(* CODESYS project lab1.project

Project tree, tasks and I/O mapping:
  Device : CODESYS Control Win V3, 3S - Smart Software Solutions GmbH, order no. 305021, version 3.5.5.50
    application Application
      libraries: Standard, * (System)
      task MainTask (cyclic, interval t#400ms, priority 1) calls task_relay
      task VISU_TASK (cyclic, interval 100 ms, priority 31) calls VisuElems.Visu_Prg
      program task_relay [ST]
      global variables GVL
      visualisation Visualization
  text list GlobalTextList
*)

// Device/Application/GVL
VAR_GLOBAL
	tempeture_sensor: INT := 20;
	door: BOOL := FALSE; // FALSE--> closed ; TRUE --> open
	
//	valve_prop: INT := -24; // FALSE--> closed ; TRUE --> open
//	btn: BOOL := FALSE; // FALSE--> closed ; TRUE --> open
//	btn_peiod: BOOL := FALSE; // FALSE--> closed ; TRUE --> open
END_VAR

// Device/Application/task_relay
PROGRAM task_relay
VAR
	DOOR_LIMIT: INT := 28;
	MIN_VALUE: INT := 15;
	MAX_VALUE: INT := 40;
	MIN_LIMIT: INT;
END_VAR

IF tempeture_sensor > DOOR_LIMIT THEN
	door:= TRUE;
ELSE door:= FALSE;
END_IF

END_PROGRAM

// Device/Application/Visualization
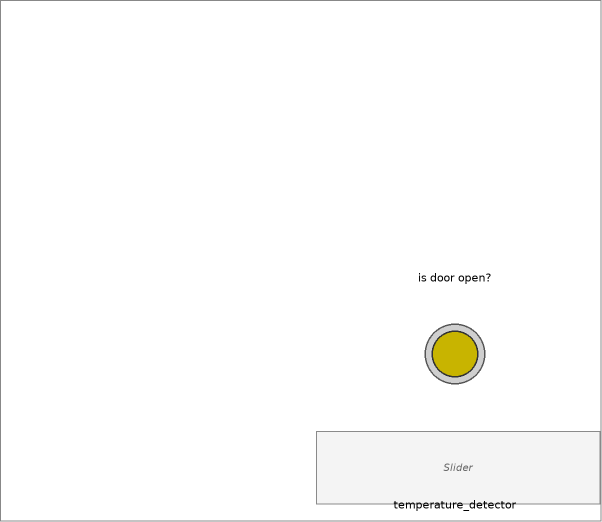
VISUALIZATION Visualization  // 602x522
    Slider (316,431 284x73), variable: tempeture_sensor, scale 15..40
    Label (380,490 150x30), "temperature_detector"
    Lamp1 (420,319 70x70), variable: door, style: Lamp-Lamp1-Yellow
    Label (380,263 150x30), "is door open?"
END_VISUALIZATION
